(* IEC 61131-3 sources: repolevel_ST_code_completion/dataset/project_code/four-level_elevator_control/FUN, 3 files *)

(* ---- F_CheckJobInDirection.st ---- *)
FUNCTION F_CheckJobInDirection : BOOL
VAR_INPUT
	nStartFloor		:	USINT;		//起始楼层
	nEndFloor		:	USINT;		//结束楼层
	bIncreasing		:	BOOL;		//TRUE=向上检查（递增），FALSE=向下检查（递减）
END_VAR
VAR
	i	:	USINT;
END_VAR

// 检查从起始楼层到结束楼层之间是否有电梯需要停靠的楼层
F_CheckJobInDirection := FALSE;

IF bIncreasing THEN
	// 向上检查（从低楼层到高楼层）
	FOR i := nStartFloor TO nEndFloor DO
		IF Tar_Dir.IsStopFloor[i] THEN
			F_CheckJobInDirection := TRUE;
			RETURN;
		END_IF
	END_FOR
ELSE
	// 向下检查（从高楼层到低楼层）
	FOR i := nEndFloor TO nStartFloor BY -1 DO
		IF Tar_Dir.IsStopFloor[i] THEN
			F_CheckJobInDirection := TRUE;
			RETURN;
		END_IF
	END_FOR
END_IF

(* ---- F_ClearFloorStop.st ---- *)
FUNCTION F_ClearFloorStop
VAR_INPUT
	nFloor			:	USINT;		//楼层号
	bClearUpStop	:	BOOL;		//是否清除上升停靠标志
	bClearDownStop	:	BOOL;		//是否清除下降停靠标志
	bClearStopFloor	:	BOOL;		//是否清除楼层停靠标志
END_VAR

// 清除楼层停靠标志
IF bClearUpStop AND (nFloor <= MaxNumFloor - 1) THEN
	Tar_Dir.IsUpStop[nFloor] := FALSE;
	QFloorUpLed[nFloor] := FALSE;
END_IF

IF bClearDownStop AND (nFloor >= 2) THEN
	Tar_Dir.IsDownStop[nFloor] := FALSE;
	QFloorDownLed[nFloor] := FALSE;
END_IF

IF bClearStopFloor THEN
	Tar_Dir.IsStopFloor[nFloor] := FALSE;
END_IF

// 清除电梯内按钮LED
IF bClearStopFloor THEN
	QGoFloorLed[nFloor] := FALSE;
END_IF

(* ---- F_SetElevatorDirection.st ---- *)
FUNCTION F_SetElevatorDirection
VAR_INPUT
	nCurrentFloor	:	USINT;		//当前楼层
	nTargetFloor	:	USINT;		//目标楼层
END_VAR

// 根据当前楼层和目标楼层设定电梯运行方向
IF nTargetFloor > nCurrentFloor THEN
	// 目标楼层高于当前楼层，电梯上升
	Tar_Dir.IsPositive := TRUE;
	Tar_Dir.IsNegative := FALSE;
ELSIF nTargetFloor < nCurrentFloor THEN
	// 目标楼层低于当前楼层，电梯下降
	Tar_Dir.IsPositive := FALSE;
	Tar_Dir.IsNegative := TRUE;
END_IF
// 如果目标楼层等于当前楼层，不改变方向
